{attribute 'qualified_only'}
VAR_GLOBAL
	// Safety Error Condition
	Error		AT%I*:	BOOL;
	// Run/Stop Safety
	Run			AT%Q*:	BOOL;
	// Restart Safety
	Restart		AT%Q*:	BOOL;
	// Error Acknowledgement 
	ErrAck		AT%Q*:	BOOL;
	// Stop signal coming from Safety
	// Stop		AT%I*:	BOOL;
	// state variable
	State		AT%I*:	USINT;
	
	Reset_STO_Azimuth		AT%Q*: BOOL;
	Reset_STO_Elevation		AT%Q*: BOOL;
	Reset_STO_Derotator		AT%Q*: BOOL;
END_VAR

(* stored: Version 1.1.0.1, ProductVersion 3.1.4024.12
   GVL GVL_Safety: Id {caac09d8-917a-47af-9e38-03ae3a5a9ed5} *)
